TYPE csp_transfer_main_statistics_debug_struct :
STRUCT
	step_id:				INT;
	reject_reason:			DWORD;
	status:					DWORD;
	//item_has:				INT;
END_STRUCT
END_TYPE

(* stored: Version 1.1.0.1, ProductVersion 3.1.4022.12
   DUT csp_transfer_main_statistics_debug_struct: Id {ff52f87a-d54e-42fe-a7c0-a42e2e7c8b29} *)
